PROGRAM ABB_Control_FB
VAR_INPUT
	mxScan: BOOL;
	qxCon1: BOOL;
	mxCon_1_ATtableScan: BOOL;
	qxCon2: BOOL;
	mxCon_2_ATtableScan: BOOL;
	qxCon3: BOOL;
	mxCon_3_ATtableScan: BOOL;
	qxPart_1_Assemble: BOOL;
	qxPart_2_Assemble: BOOL;
	qxPart_3_Assemble: BOOL;
	ixGoTo_AGV: BOOL;
	qxScanBuffer_1: BOOL;
	qxScanBuffer_2: BOOL;
	qxScanBuffer_3: BOOL;
	qxAssemblyDone: BOOL;
	mxConLeave: BOOL;
	qxGotoHome: BOOL;
	ixGotoHome: BOOL;
	qxGotoTable: BOOL;
	ixGotoTable: BOOL;
	qxGotoAGV: BOOL;
	ixGotoAGV: BOOL;
	qxGotoScanner: BOOL;
	ixGotoScanner: BOOL;
	qxGotoBuffer: BOOL;
	ixGotoBuffer: BOOL;
	qxPickBuffer1: BOOL;
	ixPickBuffer1: BOOL;
	qxPickBuffer2: BOOL;
	ixPickBuffer2: BOOL;
	qxPickBuffer3: BOOL;
	ixPickBuffer3: BOOL;
	qxLeaveBuffer1: BOOL;
	ixLeaveBuffer1: BOOL;
	qxLeaveBuffer2: BOOL;
	ixLeaveBuffer2: BOOL;
	qxLeaveBuffer3: BOOL;
	ixLeaveBuffer3: BOOL;
	qxPickScanner: BOOL;
	ixPickScanner: BOOL;
	qxLeaveScanner: BOOL;
	ixLeaveScanner: BOOL;
	qxPickAGV: BOOL;
	ixPickAGV: BOOL;
	qxLeaveAGV: BOOL;
	ixLeaveAGV: BOOL;
	qxPickTable: BOOL;
	ixPickTable: BOOL;
	qxLeaveTable: BOOL;
	ixLeaveTable: BOOL;
	ixScanBuffer: BOOL;
	ixScanContainer: BOOL;
	ixScanPart1: BOOL;
	ixScanPart2: BOOL;
	ixScanPart3: BOOL;
	ixAssemble1: BOOL;
	ixAssemble2: BOOL;
	ixAssemble3: BOOL;
	ixSendOrder: BOOL;
	ixFinishOrder: BOOL;
	mxAsse_1_done: BOOL;
	mxAsse_2_done: BOOL;
	mxAsse_3_done: BOOL;
END_VAR

VAR
	ABBGotoHome_1: ABBGotoHome;
	Auto_Mode: RS;
	Manual_Mode: RS;
	ABBGotoBufferPick_1: ABBGotoBuffer;
	ABBPickLeaveBufferPick_1: ABBPickLeaveBuffer;
	ABBGotoScanner_1: ABBGotoScanner;
	ABBPickLeaveScannerLB_1: ABBPickLeaveScanner;
	SensorReader_buffer_1: SensorReader;
	ABBScannerStation_1: ABBScannerStation;
	ABBPickLeaveScannerPB_1: ABBPickLeaveScanner;
	ABBGotoBufferLeave_1: ABBGotoBuffer;
	ABBPickLeaveBufferLeave_1: ABBPickLeaveBuffer;
	mxBuffer_1_scanned: BOOL;
	Reading_1_Done: RS;
	ABBGotoBufferPick_2: ABBGotoBuffer;
	ABBPickLeaveBufferPick_2: ABBPickLeaveBuffer;
	ABBGotoScanner_2: ABBGotoScanner;
	ABBPickLeaveScannerLB_2: ABBPickLeaveScanner;
	ABBScannerStation_2: ABBScannerStation;
	ABBPickLeaveScannerPB_2: ABBPickLeaveScanner;
	ABBGotoBufferLeave_2: ABBGotoBuffer;
	ABBPickLeaveBufferLeave_2: ABBPickLeaveBuffer;
	mxBuffer_2_scanned: BOOL;
	ABBGotoBufferPick_3: ABBGotoBuffer;
	ABBPickLeaveBufferPick_3: ABBPickLeaveBuffer;
	ABBGotoScanner_3: ABBGotoScanner;
	ABBPickLeaveScannerLB_3: ABBPickLeaveScanner;
	ABBScannerStation_3: ABBScannerStation;
	ABBPickLeaveScannerPB_3: ABBPickLeaveScanner;
	ABBGotoBufferLeave_3: ABBGotoBuffer;
	ABBPickLeaveBufferLeave_3: ABBPickLeaveBuffer;
	mxBuffer_3_scanned: BOOL;
	ABBGotoHome_AGV_Con1: ABBGotoHome;
	SensorReader_0: SensorReader;
	Scanner_FB_0: Scanner_FB;
	mxRP: BOOL;
	mxYP: BOOL;
	mxBP: BOOL;
	mxRCy: BOOL;
	mxYCy: BOOL;
	mxBCy: BOOL;
	mxYOct: BOOL;
	mxBOct: BOOL;
	mxROct: BOOL;
	mxIP: BOOL;
	Sensor_Sense_0: Sensor_Sense;
	mxRCon: BOOL;
	mxYCon: BOOL;
	mxBCon: BOOL;
	mxContainerScanDone: BOOL;
	mxScanner: BOOL;
	Scan_Block: RS;
	mxScanDone: BOOL;
	ABBGotoAGVPos_1: ABBGotoAGVPos;
	ABBPickLeaveContainerAGV_1: ABBPickLeaveContainerAGV;
	ABBGotoScannerCon_1: ABBGotoScanner;
	ABBPickLeaveContainerAGVPick_1: ABBPickLeaveContainerAGV;
	ABBPickLeaveContainerAGVLeave_1: ABBPickLeaveContainerAGV;
	ABBPickLeaveScannerLC_1: ABBPickLeaveScanner;
	ABBScanContainer_1: ABBScanContainer;
	ABBScannerStationCon1_1: ABBScannerStation;
	ABBPickLeaveScannerPC_1: ABBPickLeaveScanner;
	ABBGotoTableCon_1: ABBGotoTable;
	ABBGotoTableCon_1_Scanned: ABBGotoTable;
	ABBGotoTableCon_2: ABBGotoTable;
	ABBScanContainer_2: ABBScanContainer;
	ABBGotoTableCon_2_Scanned: ABBGotoTable;
	ABBGotoTableCon_3: ABBGotoTable;
	ABBScanContainer_3: ABBScanContainer;
	ABBGotoTableCon_3_Scanned: ABBGotoTable;
	ABBAssemble_1: ABBAssemble;
	ABBGotoTable_Ass1: ABBGotoTable;
	
	ABBAssemble_2: ABBAssemble;
	ABBGotoTable_Ass2: ABBGotoTable;
	
	ABBAssemble_3: ABBAssemble;
	ABBGotoTable_Ass3: ABBGotoTable;
	
	TON_0: TON;
	ABBPickLeaveContaineronTableLeave_1: ABBPickLeaveContaineronTable;
	ABBPickLeaveContaineronTableLeave_2: ABBPickLeaveContaineronTable;
	ABBPickLeaveContaineronTableLeave_3: ABBPickLeaveContaineronTable;
	ABBGotoTable_0: ABBGotoTable;
	ABBPickLeaveContaineronTableLeave_0: ABBPickLeaveContaineronTable;
	TON_1: TON;
	TON_2: TON;
	TON_3: TON;
	ABBGotoTable_Assembled: ABBGotoTable;
	ABBPickLeaveContaineronTable_Assembled: ABBPickLeaveContaineronTable;
	ABBGotoAGVPos_Assembled: ABBGotoAGVPos;
	ABBPickLeaveContainerAGV_Assembled: ABBPickLeaveContainerAGV;
	ABBAssemble_Part1: ABBAssemble;
	ABBAssemble_Part2: ABBAssemble;
	ABBAssemble_Part3: ABBAssemble;
	ABBGotoHome_Next_Assemnbly: ABBGotoHome;
	mxWaitforNext: BOOL;
	ABBGotoHome_10: ABBGotoHome;
	qxHOME: BOOL;
	ABBGotoTable_10: ABBGotoTable;
	qxTABLE: BOOL;
	ABBGotoAGVPos_10: ABBGotoAGVPos;
	qxAGV: BOOL;
	ABBGotoScanner_10: ABBGotoScanner;
	qxSCANNER: BOOL;
	ABBGotoBuffer_10: ABBGotoBuffer;
	qxBUFFER: BOOL;
	ABBPickLeaveBuffer_Pick: ABBPickLeaveBuffer;
	qxBufferPicked1: BOOL;
	ABBPickLeaveBuffer_Leave: ABBPickLeaveBuffer;
	qxBufferLeft1: BOOL;
	ABBGotoScanner_Pick: ABBGotoScanner;
	ABBPickLeaveScanner_Pick: ABBPickLeaveScanner;
	qxPickedScanner: BOOL;
	ABBGotoScanner_Leave: ABBGotoScanner;
	ABBPickLeaveScanner_Leave: ABBPickLeaveScanner;
	qxLeftScanner: BOOL;
	ABBGotoAGVPos_Pick: ABBGotoAGVPos;
	ABBPickLeaveContainerAGV_Pick: ABBPickLeaveContainerAGV;
	qxPickedAGV: BOOL;
	ABBGotoAGVPos_Leave: ABBGotoAGVPos;
	ABBPickLeaveContainerAGV_Leave: ABBPickLeaveContainerAGV;
	qxLeftAGV: BOOL;
	ABBGotoTable_Pick: ABBGotoTable;
	ABBPickLeaveContaineronTable_Pick: ABBPickLeaveContaineronTable;
	qxPickedTable: BOOL;
	ABBGotoTable_Leave: ABBGotoTable;
	ABBPickLeaveContaineronTable_Leave: ABBPickLeaveContaineronTable;
	qxLeftTable: BOOL;
END_VAR
VAR // added by the converter: edge detectors and wires of the graphical bodies
    _w1, _w2, _w3, _w4, _w5, _w6, _w7 : BOOL;
END_VAR

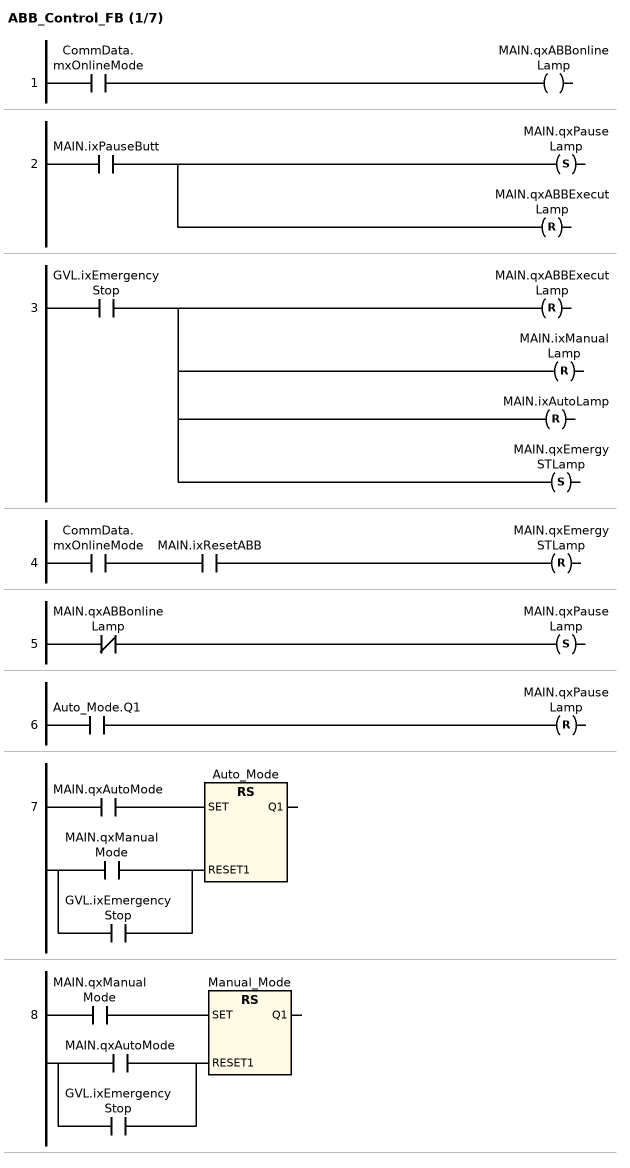
// NETWORK 1
MAIN.qxABBonlineLamp := CommData.mxOnlineMode;

// NETWORK 2
_w1 := MAIN.ixPauseButt;
MAIN.qxPauseLamp S= _w1;
MAIN.qxABBExecutLamp R= _w1;

// NETWORK 3
MAIN.qxABBExecutLamp R= GVL.ixEmergencyStop;
MAIN.ixManualLamp R= GVL.ixEmergencyStop;
MAIN.ixAutoLamp R= GVL.ixEmergencyStop;
MAIN.qxEmergySTLamp S= GVL.ixEmergencyStop;

// NETWORK 4
MAIN.qxEmergySTLamp R= CommData.mxOnlineMode AND MAIN.ixResetABB;

// NETWORK 5
MAIN.qxPauseLamp S= NOT MAIN.qxABBonlineLamp;

// NETWORK 6
MAIN.qxPauseLamp R= Auto_Mode.Q1;

// NETWORK 7
Auto_Mode(SET := MAIN.qxAutoMode, RESET1 := MAIN.qxManualMode OR GVL.ixEmergencyStop); // RS

// NETWORK 8
Manual_Mode(SET := MAIN.qxManualMode, RESET1 := MAIN.qxAutoMode OR GVL.ixEmergencyStop); // RS

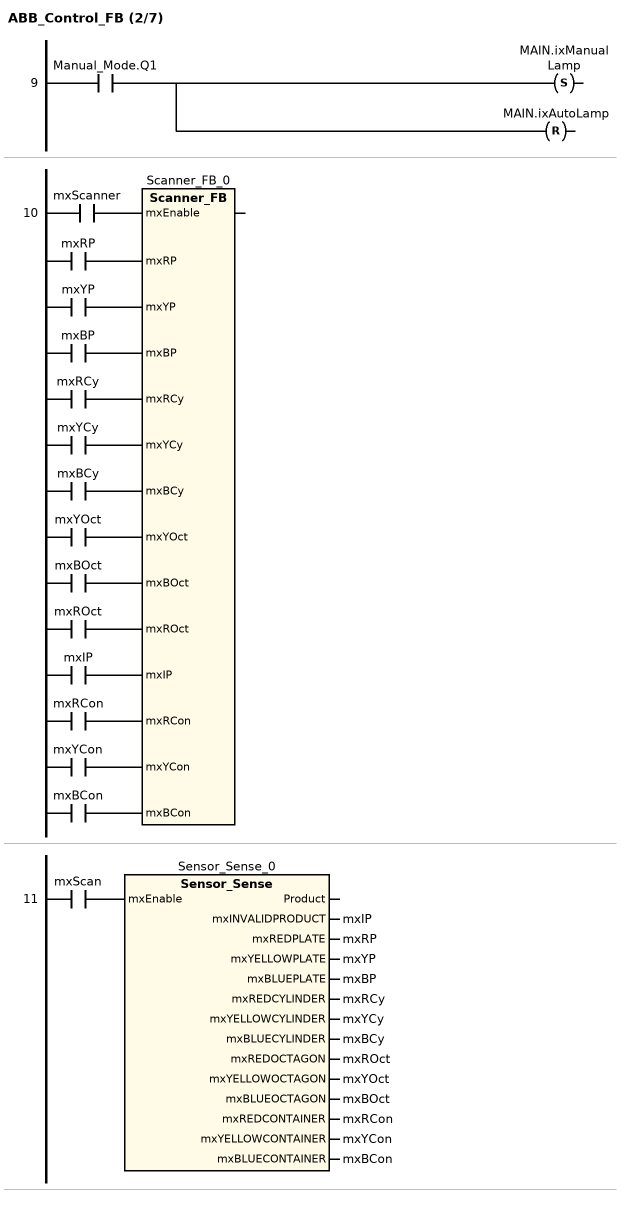
// NETWORK 9
MAIN.ixManualLamp S= Manual_Mode.Q1;
MAIN.ixAutoLamp R= Manual_Mode.Q1;

// NETWORK 10
Scanner_FB_0(
    mxEnable := mxScanner,
    mxRP := mxRP,
    mxYP := mxYP,
    mxBP := mxBP,
    mxRCy := mxRCy,
    mxYCy := mxYCy,
    mxBCy := mxBCy,
    mxYOct := mxYOct,
    mxBOct := mxBOct,
    mxROct := mxROct,
    mxIP := mxIP,
    mxRCon := mxRCon,
    mxYCon := mxYCon,
    mxBCon := mxBCon); // Scanner_FB

// NETWORK 11
Sensor_Sense_0(
    mxEnable := mxScan,
    mxINVALIDPRODUCT => mxIP,
    mxREDPLATE => mxRP,
    mxYELLOWPLATE => mxYP,
    mxBLUEPLATE => mxBP,
    mxREDCYLINDER => mxRCy,
    mxYELLOWCYLINDER => mxYCy,
    mxBLUECYLINDER => mxBCy,
    mxREDOCTAGON => mxROct,
    mxYELLOWOCTAGON => mxYOct,
    mxBLUEOCTAGON => mxBOct,
    mxREDCONTAINER => mxRCon,
    mxYELLOWCONTAINER => mxYCon,
    mxBLUECONTAINER => mxBCon); // Sensor_Sense

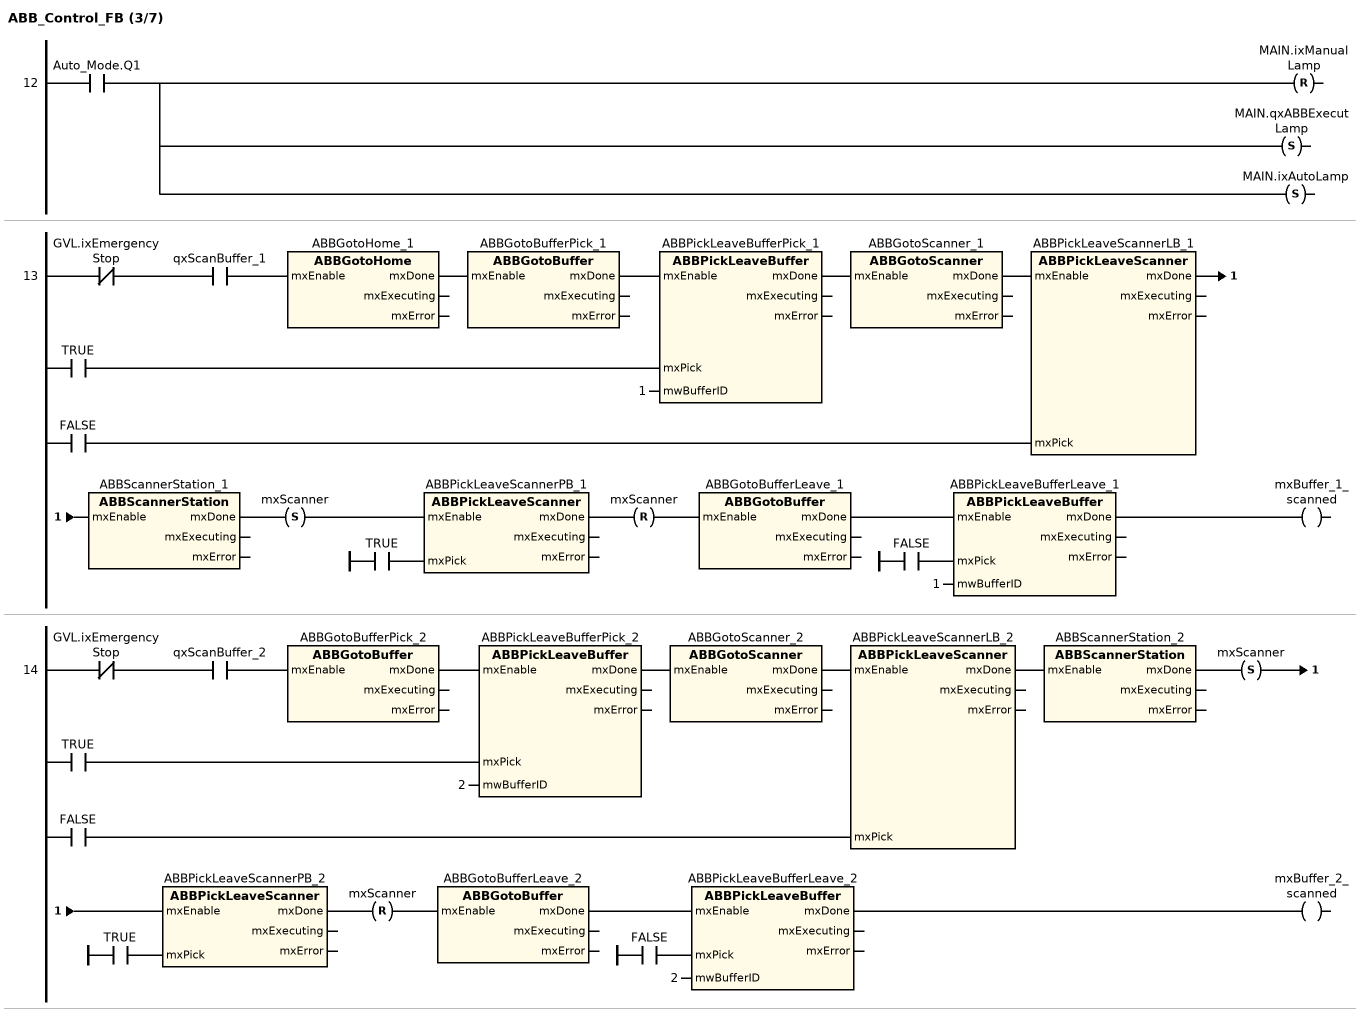
// NETWORK 12
MAIN.ixManualLamp R= Auto_Mode.Q1;
MAIN.qxABBExecutLamp S= Auto_Mode.Q1;
MAIN.ixAutoLamp S= Auto_Mode.Q1;

// NETWORK 13
ABBGotoHome_1(mxEnable := NOT GVL.ixEmergencyStop AND qxScanBuffer_1); // ABBGotoHome
ABBGotoBufferPick_1(mxEnable := ABBGotoHome_1.mxDone); // ABBGotoBuffer
ABBPickLeaveBufferPick_1(mxEnable := ABBGotoBufferPick_1.mxDone, mxPick := TRUE, mwBufferID := 1); // ABBPickLeaveBuffer
ABBGotoScanner_1(mxEnable := ABBPickLeaveBufferPick_1.mxDone); // ABBGotoScanner
ABBPickLeaveScannerLB_1(mxEnable := ABBGotoScanner_1.mxDone, mxPick := FALSE); // ABBPickLeaveScanner
ABBScannerStation_1(mxEnable := ABBPickLeaveScannerLB_1.mxDone); // ABBScannerStation
mxScanner S= ABBScannerStation_1.mxDone;
ABBPickLeaveScannerPB_1(mxEnable := ABBScannerStation_1.mxDone, mxPick := TRUE); // ABBPickLeaveScanner
mxScanner R= ABBPickLeaveScannerPB_1.mxDone;
ABBGotoBufferLeave_1(mxEnable := ABBPickLeaveScannerPB_1.mxDone); // ABBGotoBuffer
ABBPickLeaveBufferLeave_1(mxEnable := ABBGotoBufferLeave_1.mxDone, mxPick := FALSE, mwBufferID := 1); // ABBPickLeaveBuffer
mxBuffer_1_scanned := ABBPickLeaveBufferLeave_1.mxDone;

// NETWORK 14
ABBGotoBufferPick_2(mxEnable := NOT GVL.ixEmergencyStop AND qxScanBuffer_2); // ABBGotoBuffer
ABBPickLeaveBufferPick_2(mxEnable := ABBGotoBufferPick_2.mxDone, mxPick := TRUE, mwBufferID := 2); // ABBPickLeaveBuffer
ABBGotoScanner_2(mxEnable := ABBPickLeaveBufferPick_2.mxDone); // ABBGotoScanner
ABBPickLeaveScannerLB_2(mxEnable := ABBGotoScanner_2.mxDone, mxPick := FALSE); // ABBPickLeaveScanner
ABBScannerStation_2(mxEnable := ABBPickLeaveScannerLB_2.mxDone); // ABBScannerStation
mxScanner S= ABBScannerStation_2.mxDone;
ABBPickLeaveScannerPB_2(mxEnable := ABBScannerStation_2.mxDone, mxPick := TRUE); // ABBPickLeaveScanner
mxScanner R= ABBPickLeaveScannerPB_2.mxDone;
ABBGotoBufferLeave_2(mxEnable := ABBPickLeaveScannerPB_2.mxDone); // ABBGotoBuffer
ABBPickLeaveBufferLeave_2(mxEnable := ABBGotoBufferLeave_2.mxDone, mxPick := FALSE, mwBufferID := 2); // ABBPickLeaveBuffer
mxBuffer_2_scanned := ABBPickLeaveBufferLeave_2.mxDone;

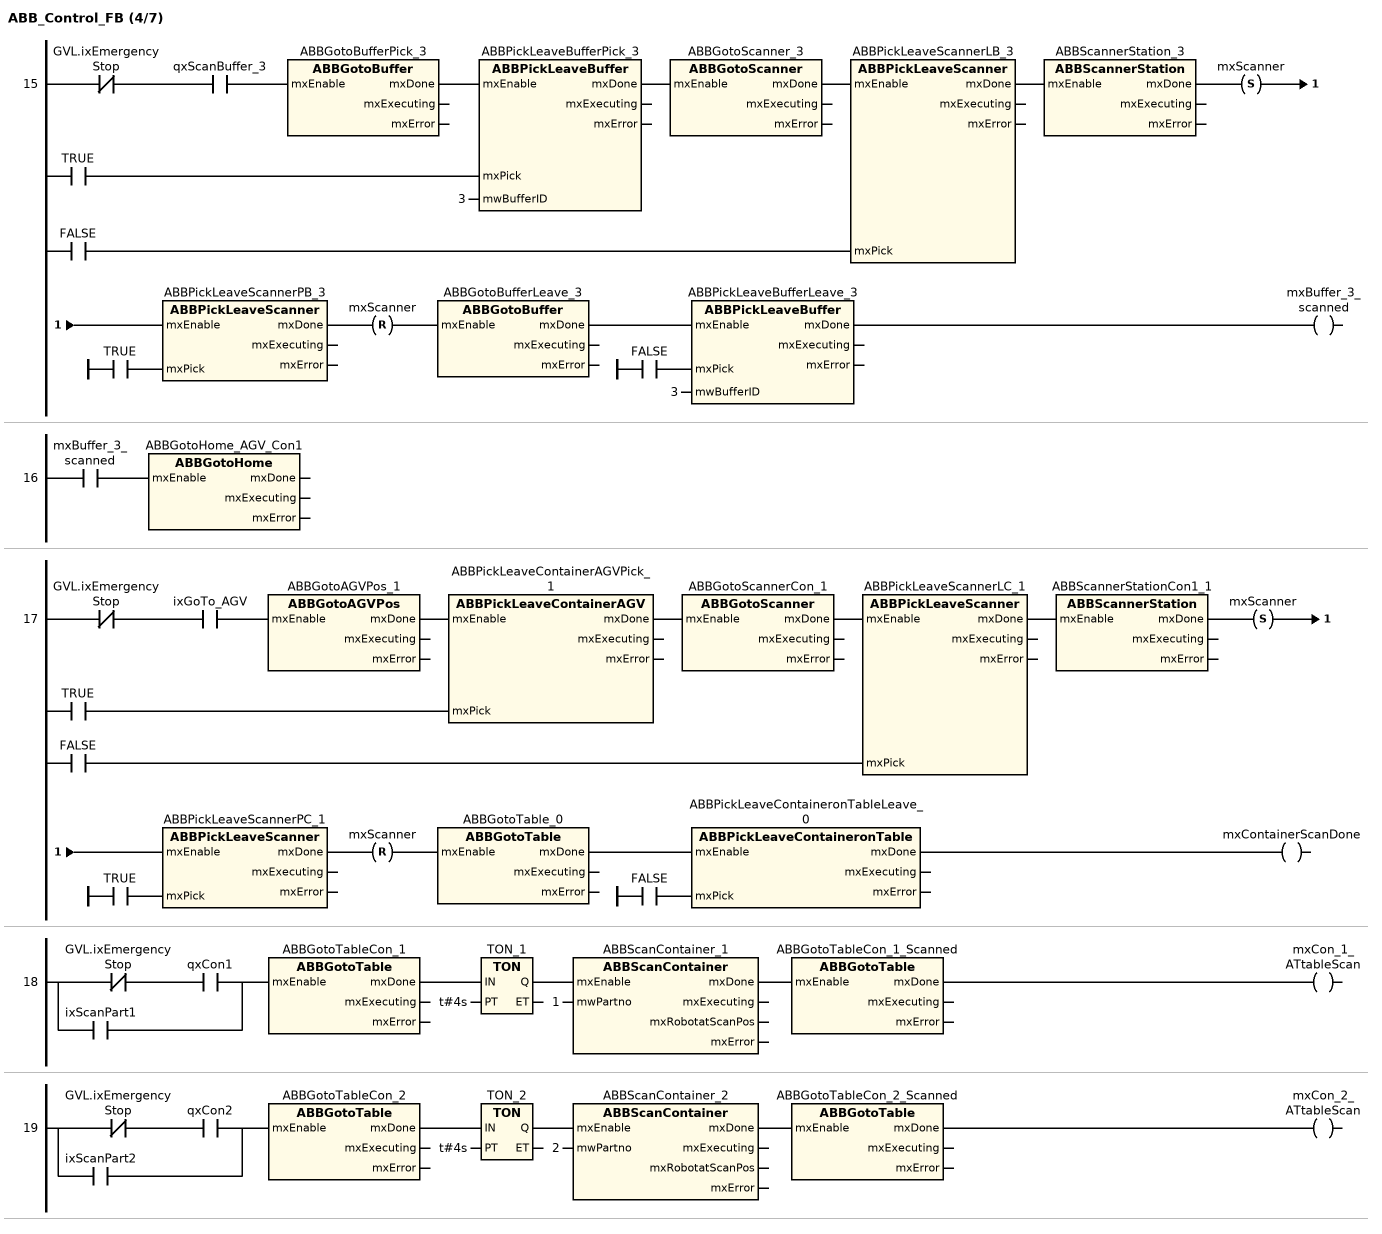
// NETWORK 15
ABBGotoBufferPick_3(mxEnable := NOT GVL.ixEmergencyStop AND qxScanBuffer_3); // ABBGotoBuffer
ABBPickLeaveBufferPick_3(mxEnable := ABBGotoBufferPick_3.mxDone, mxPick := TRUE, mwBufferID := 3); // ABBPickLeaveBuffer
ABBGotoScanner_3(mxEnable := ABBPickLeaveBufferPick_3.mxDone); // ABBGotoScanner
ABBPickLeaveScannerLB_3(mxEnable := ABBGotoScanner_3.mxDone, mxPick := FALSE); // ABBPickLeaveScanner
ABBScannerStation_3(mxEnable := ABBPickLeaveScannerLB_3.mxDone); // ABBScannerStation
mxScanner S= ABBScannerStation_3.mxDone;
ABBPickLeaveScannerPB_3(mxEnable := ABBScannerStation_3.mxDone, mxPick := TRUE); // ABBPickLeaveScanner
mxScanner R= ABBPickLeaveScannerPB_3.mxDone;
ABBGotoBufferLeave_3(mxEnable := ABBPickLeaveScannerPB_3.mxDone); // ABBGotoBuffer
ABBPickLeaveBufferLeave_3(mxEnable := ABBGotoBufferLeave_3.mxDone, mxPick := FALSE, mwBufferID := 3); // ABBPickLeaveBuffer
mxBuffer_3_scanned := ABBPickLeaveBufferLeave_3.mxDone;

// NETWORK 16
ABBGotoHome_AGV_Con1(mxEnable := mxBuffer_3_scanned); // ABBGotoHome

// NETWORK 17
ABBGotoAGVPos_1(mxEnable := NOT GVL.ixEmergencyStop AND ixGoTo_AGV); // ABBGotoAGVPos
ABBPickLeaveContainerAGVPick_1(mxEnable := ABBGotoAGVPos_1.mxDone, mxPick := TRUE); // ABBPickLeaveContainerAGV
ABBGotoScannerCon_1(mxEnable := ABBPickLeaveContainerAGVPick_1.mxDone); // ABBGotoScanner
ABBPickLeaveScannerLC_1(mxEnable := ABBGotoScannerCon_1.mxDone, mxPick := FALSE); // ABBPickLeaveScanner
ABBScannerStationCon1_1(mxEnable := ABBPickLeaveScannerLC_1.mxDone); // ABBScannerStation
mxScanner S= ABBScannerStationCon1_1.mxDone;
ABBPickLeaveScannerPC_1(mxEnable := ABBScannerStationCon1_1.mxDone, mxPick := TRUE); // ABBPickLeaveScanner
mxScanner R= ABBPickLeaveScannerPC_1.mxDone;
ABBGotoTable_0(mxEnable := ABBPickLeaveScannerPC_1.mxDone); // ABBGotoTable
ABBPickLeaveContaineronTableLeave_0(mxEnable := ABBGotoTable_0.mxDone, mxPick := FALSE); // ABBPickLeaveContaineronTable
mxContainerScanDone := ABBPickLeaveContaineronTableLeave_0.mxDone;

// NETWORK 18
ABBGotoTableCon_1(mxEnable := NOT GVL.ixEmergencyStop AND qxCon1 OR ixScanPart1); // ABBGotoTable
TON_1(IN := ABBGotoTableCon_1.mxDone, PT := t#4s); // TON
ABBScanContainer_1(mxEnable := TON_1.Q, mwPartno := 1); // ABBScanContainer
ABBGotoTableCon_1_Scanned(mxEnable := ABBScanContainer_1.mxDone); // ABBGotoTable
mxCon_1_ATtableScan := ABBGotoTableCon_1_Scanned.mxDone;

// NETWORK 19
ABBGotoTableCon_2(mxEnable := NOT GVL.ixEmergencyStop AND qxCon2 OR ixScanPart2); // ABBGotoTable
TON_2(IN := ABBGotoTableCon_2.mxDone, PT := t#4s); // TON
ABBScanContainer_2(mxEnable := TON_2.Q, mwPartno := 2); // ABBScanContainer
ABBGotoTableCon_2_Scanned(mxEnable := ABBScanContainer_2.mxDone); // ABBGotoTable
mxCon_2_ATtableScan := ABBGotoTableCon_2_Scanned.mxDone;

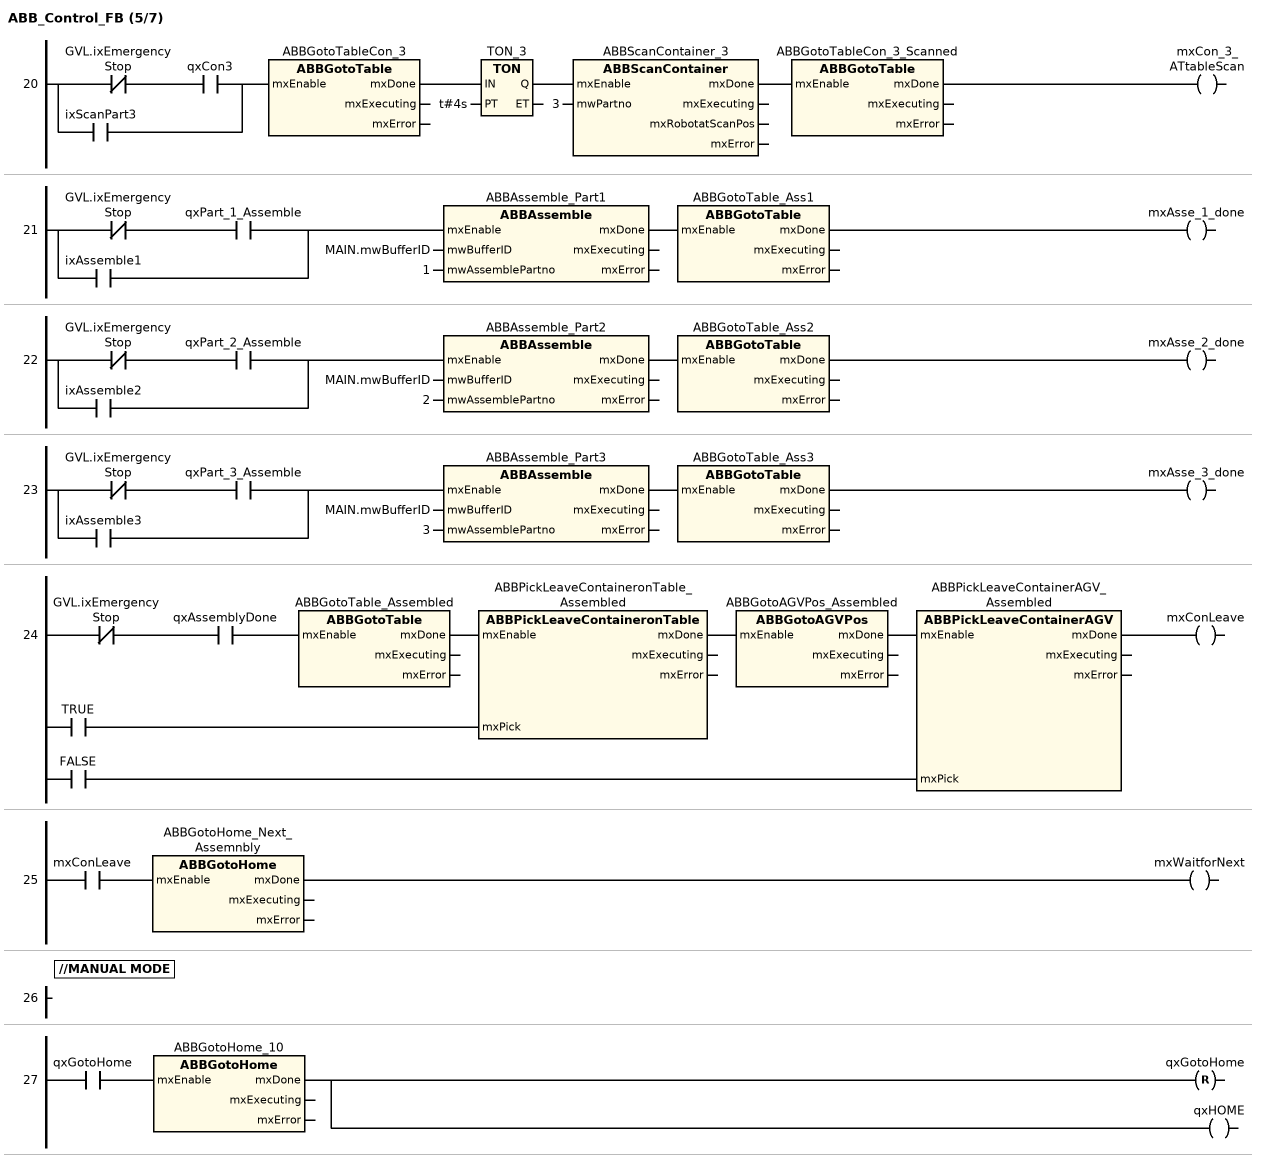
// NETWORK 20
ABBGotoTableCon_3(mxEnable := NOT GVL.ixEmergencyStop AND qxCon3 OR ixScanPart3); // ABBGotoTable
TON_3(IN := ABBGotoTableCon_3.mxDone, PT := t#4s); // TON
ABBScanContainer_3(mxEnable := TON_3.Q, mwPartno := 3); // ABBScanContainer
ABBGotoTableCon_3_Scanned(mxEnable := ABBScanContainer_3.mxDone); // ABBGotoTable
mxCon_3_ATtableScan := ABBGotoTableCon_3_Scanned.mxDone;

// NETWORK 21
ABBAssemble_Part1(
    mxEnable := NOT GVL.ixEmergencyStop AND qxPart_1_Assemble OR ixAssemble1,
    mwBufferID := MAIN.mwBufferID,
    mwAssemblePartno := 1); // ABBAssemble
ABBGotoTable_Ass1(mxEnable := ABBAssemble_Part1.mxDone); // ABBGotoTable
mxAsse_1_done := ABBGotoTable_Ass1.mxDone;

// NETWORK 22
ABBAssemble_Part2(
    mxEnable := NOT GVL.ixEmergencyStop AND qxPart_2_Assemble OR ixAssemble2,
    mwBufferID := MAIN.mwBufferID,
    mwAssemblePartno := 2); // ABBAssemble
ABBGotoTable_Ass2(mxEnable := ABBAssemble_Part2.mxDone); // ABBGotoTable
mxAsse_2_done := ABBGotoTable_Ass2.mxDone;

// NETWORK 23
ABBAssemble_Part3(
    mxEnable := NOT GVL.ixEmergencyStop AND qxPart_3_Assemble OR ixAssemble3,
    mwBufferID := MAIN.mwBufferID,
    mwAssemblePartno := 3); // ABBAssemble
ABBGotoTable_Ass3(mxEnable := ABBAssemble_Part3.mxDone); // ABBGotoTable
mxAsse_3_done := ABBGotoTable_Ass3.mxDone;

// NETWORK 24
ABBGotoTable_Assembled(mxEnable := NOT GVL.ixEmergencyStop AND qxAssemblyDone); // ABBGotoTable
ABBPickLeaveContaineronTable_Assembled(mxEnable := ABBGotoTable_Assembled.mxDone, mxPick := TRUE); // ABBPickLeaveContaineronTable
ABBGotoAGVPos_Assembled(mxEnable := ABBPickLeaveContaineronTable_Assembled.mxDone); // ABBGotoAGVPos
ABBPickLeaveContainerAGV_Assembled(mxEnable := ABBGotoAGVPos_Assembled.mxDone, mxPick := FALSE); // ABBPickLeaveContainerAGV
mxConLeave := ABBPickLeaveContainerAGV_Assembled.mxDone;

// NETWORK 25
ABBGotoHome_Next_Assemnbly(mxEnable := mxConLeave); // ABBGotoHome
mxWaitforNext := ABBGotoHome_Next_Assemnbly.mxDone;

// NETWORK 26
// label: //MANUAL MODE

// NETWORK 27
ABBGotoHome_10(mxEnable := qxGotoHome); // ABBGotoHome
qxGotoHome R= ABBGotoHome_10.mxDone;
qxHOME := ABBGotoHome_10.mxDone;

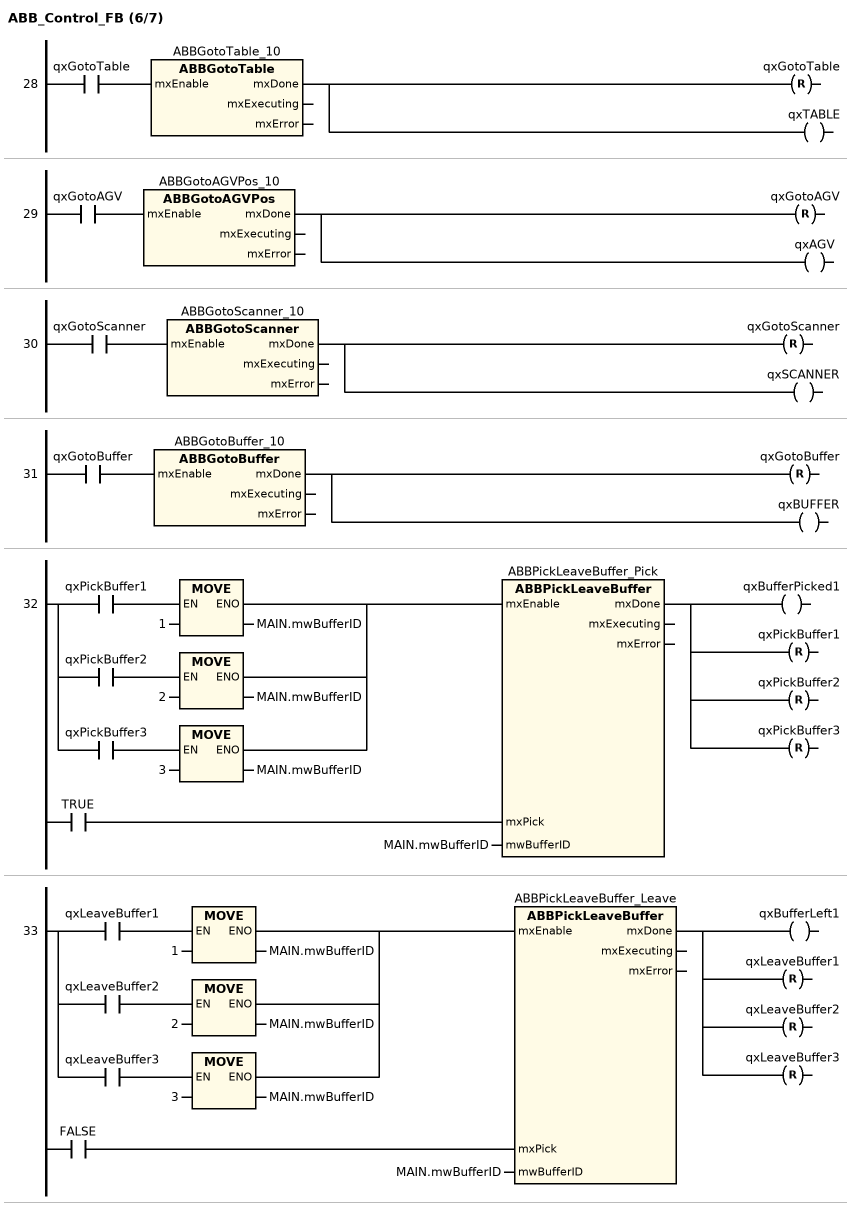
// NETWORK 28
ABBGotoTable_10(mxEnable := qxGotoTable); // ABBGotoTable
qxGotoTable R= ABBGotoTable_10.mxDone;
qxTABLE := ABBGotoTable_10.mxDone;

// NETWORK 29
ABBGotoAGVPos_10(mxEnable := qxGotoAGV); // ABBGotoAGVPos
qxGotoAGV R= ABBGotoAGVPos_10.mxDone;
qxAGV := ABBGotoAGVPos_10.mxDone;

// NETWORK 30
ABBGotoScanner_10(mxEnable := qxGotoScanner); // ABBGotoScanner
qxGotoScanner R= ABBGotoScanner_10.mxDone;
qxSCANNER := ABBGotoScanner_10.mxDone;

// NETWORK 31
ABBGotoBuffer_10(mxEnable := qxGotoBuffer); // ABBGotoBuffer
qxGotoBuffer R= ABBGotoBuffer_10.mxDone;
qxBUFFER := ABBGotoBuffer_10.mxDone;

// NETWORK 32
_w2 := qxPickBuffer1;
IF _w2 THEN MAIN.mwBufferID := 1; END_IF
_w3 := qxPickBuffer2;
IF _w3 THEN MAIN.mwBufferID := 2; END_IF
_w4 := qxPickBuffer3;
IF _w4 THEN MAIN.mwBufferID := 3; END_IF
ABBPickLeaveBuffer_Pick(mxEnable := _w2 OR _w3 OR _w4, mxPick := TRUE, mwBufferID := MAIN.mwBufferID); // ABBPickLeaveBuffer
qxBufferPicked1 := ABBPickLeaveBuffer_Pick.mxDone;
qxPickBuffer1 R= ABBPickLeaveBuffer_Pick.mxDone;
qxPickBuffer2 R= ABBPickLeaveBuffer_Pick.mxDone;
qxPickBuffer3 R= ABBPickLeaveBuffer_Pick.mxDone;

// NETWORK 33
_w5 := qxLeaveBuffer1;
IF _w5 THEN MAIN.mwBufferID := 1; END_IF
_w6 := qxLeaveBuffer2;
IF _w6 THEN MAIN.mwBufferID := 2; END_IF
_w7 := qxLeaveBuffer3;
IF _w7 THEN MAIN.mwBufferID := 3; END_IF
ABBPickLeaveBuffer_Leave(mxEnable := _w5 OR _w6 OR _w7, mxPick := FALSE, mwBufferID := MAIN.mwBufferID); // ABBPickLeaveBuffer
qxBufferLeft1 := ABBPickLeaveBuffer_Leave.mxDone;
qxLeaveBuffer1 R= ABBPickLeaveBuffer_Leave.mxDone;
qxLeaveBuffer2 R= ABBPickLeaveBuffer_Leave.mxDone;
qxLeaveBuffer3 R= ABBPickLeaveBuffer_Leave.mxDone;

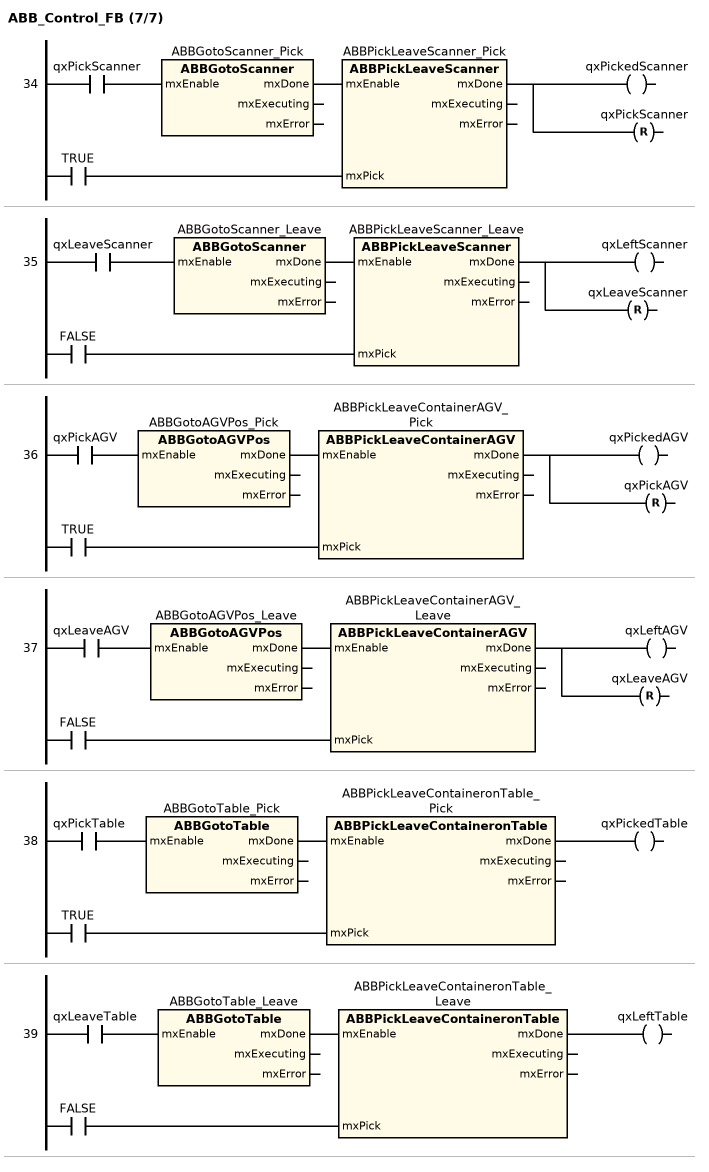
// NETWORK 34
ABBGotoScanner_Pick(mxEnable := qxPickScanner); // ABBGotoScanner
ABBPickLeaveScanner_Pick(mxEnable := ABBGotoScanner_Pick.mxDone, mxPick := TRUE); // ABBPickLeaveScanner
qxPickedScanner := ABBPickLeaveScanner_Pick.mxDone;
qxPickScanner R= ABBPickLeaveScanner_Pick.mxDone;

// NETWORK 35
ABBGotoScanner_Leave(mxEnable := qxLeaveScanner); // ABBGotoScanner
ABBPickLeaveScanner_Leave(mxEnable := ABBGotoScanner_Leave.mxDone, mxPick := FALSE); // ABBPickLeaveScanner
qxLeftScanner := ABBPickLeaveScanner_Leave.mxDone;
qxLeaveScanner R= ABBPickLeaveScanner_Leave.mxDone;

// NETWORK 36
ABBGotoAGVPos_Pick(mxEnable := qxPickAGV); // ABBGotoAGVPos
ABBPickLeaveContainerAGV_Pick(mxEnable := ABBGotoAGVPos_Pick.mxDone, mxPick := TRUE); // ABBPickLeaveContainerAGV
qxPickedAGV := ABBPickLeaveContainerAGV_Pick.mxDone;
qxPickAGV R= ABBPickLeaveContainerAGV_Pick.mxDone;

// NETWORK 37
ABBGotoAGVPos_Leave(mxEnable := qxLeaveAGV); // ABBGotoAGVPos
ABBPickLeaveContainerAGV_Leave(mxEnable := ABBGotoAGVPos_Leave.mxDone, mxPick := FALSE); // ABBPickLeaveContainerAGV
qxLeftAGV := ABBPickLeaveContainerAGV_Leave.mxDone;
qxLeaveAGV R= ABBPickLeaveContainerAGV_Leave.mxDone;

// NETWORK 38
ABBGotoTable_Pick(mxEnable := qxPickTable); // ABBGotoTable
ABBPickLeaveContaineronTable_Pick(mxEnable := ABBGotoTable_Pick.mxDone, mxPick := TRUE); // ABBPickLeaveContaineronTable
qxPickedTable := ABBPickLeaveContaineronTable_Pick.mxDone;

// NETWORK 39
ABBGotoTable_Leave(mxEnable := qxLeaveTable); // ABBGotoTable
ABBPickLeaveContaineronTable_Leave(mxEnable := ABBGotoTable_Leave.mxDone, mxPick := FALSE); // ABBPickLeaveContaineronTable
qxLeftTable := ABBPickLeaveContaineronTable_Leave.mxDone;

END_PROGRAM

(* stored: Version 1.1.0.1, ProductVersion 3.1.4024.12
   POU ABB_Control_FB: Id {5dd92650-74f8-46de-90d1-5646e5a09465}, SpecialFunc None *)
